// Mitsubishi GX Works2 project: plc   PLC: FX3G

// global labels: Global1
VAR_GLOBAL CONSTANT
  reset_petel_stocks : INT;
END_VAR
VAR_GLOBAL
  petel_stocks AT D2000 : REAL;
  petel_input AT D2500 : REAL;
  lemon_stocks AT D4000 : REAL;
  lemon_input AT D4500 : REAL;
  stabilizer_stocks AT D3000 : REAL;
  stabilizer_input AT D3500 : REAL;
  gummy_stocks AT D5000 : REAL;
  gummy_input AT D5500 : REAL;
  braek_switch AT X005 : BOOL;
  start_switch AT X007 : BOOL;
  valid_input : BOOL;
  start_proces AT X001 : BOOL;
  analog_input AT D8280 : INT;
END_VAR
VAR_GLOBAL CONSTANT
  convert : REAL := 400;
END_VAR
VAR_GLOBAL
  analog_output AT D8282 : INT;
END_VAR
VAR_GLOBAL CONSTANT
  reset_lemonl_stocks : INT;
END_VAR
VAR_GLOBAL
  day_work AT Y007 : BOOL;
  analog_input1_sampled AT M0 : BOOL;
  save_analog_input1 AT D8200 : REAL;
END_VAR
VAR_GLOBAL CONSTANT
  max5 : REAL := 5;
  min6 : REAL := 6;
END_VAR
VAR_GLOBAL
  pinuk_check AT M1 : BOOL;
  regular_check AT M2 : BOOL;
END_VAR
VAR_GLOBAL CONSTANT
  lemon_min_regular : REAL := 455.0;
  petel_min_regular : REAL := 280.0;
  stabilizer_min_regular : REAL := 105.0;
END_VAR
VAR_GLOBAL
  can_make_regular : BOOL;
END_VAR
VAR_GLOBAL CONSTANT
  lemon_min_pinuk : REAL := 655.0;
  petel_min_pinuk : REAL := 385.0;
  stabilizer_min_pinuk : REAL := 210.0;
END_VAR
VAR_GLOBAL
  can_make_pinuk : BOOL;
  make_pinuk AT M4 : BOOL;
  make_regular AT M3 : BOOL;
END_VAR
VAR_GLOBAL CONSTANT
  lemon_for_regular : REAL := 455;
  petel_for_regular : REAL := 280;
  stabilizer_for_regular : REAL := 105;
END_VAR
VAR_GLOBAL
  ready_regular AT M5 : BOOL;
END_VAR
VAR_GLOBAL CONSTANT
  lemon_for_pinuck : REAL := 665;
END_VAR
VAR_GLOBAL
  ready_pinuk AT M6 : BOOL;
END_VAR
VAR_GLOBAL CONSTANT
  petel_for_pinuk : REAL := 385.0;
  stabilizer_for_pinuk : REAL := 210.0;
END_VAR
VAR_GLOBAL
  ice_cream_making AT TC1 : BOOL;
END_VAR
VAR_GLOBAL CONSTANT
  timer_value_5 : INT := 50;
END_VAR
VAR_GLOBAL
  end_making_ice AT TS1 : BOOL;
  making_light AT Y000 : BOOL;
  start_cooling_process AT X002 : BOOL;
  lemon_container AT D6000 : REAL;
  petel_container AT D6300 : REAL;
  petel_cooling_container AT D6800 : REAL;
  lemon_cooling_container AT D7200 : REAL;
  flavors_in_cooling_container AT M7 : BOOL;
  cooling_process_on AT Y002 : BOOL;
END_VAR
VAR_GLOBAL CONSTANT
  timer_value_8 : INT := 80;
END_VAR
VAR_GLOBAL
  temperature_sensor AT X003 : BOOL;
  end_cooling_timer AT TS2 : BOOL;
  cooling_light AT Y002 : BOOL;
  finish_cooling AT M8 : BOOL;
  end_cooling AT Y002 : BOOL;
  mixing_container AT D7400 : REAL;
END_VAR
VAR_GLOBAL CONSTANT
  gummy_for_regular : REAL := 28;
  gummy_for_pinuk : REAL := 70;
END_VAR
VAR_GLOBAL
  pinuk_mixing_starts AT M10 : BOOL;
  regular_mixing_starts AT M9 : BOOL;
  mixing_time_regular AT TC3 : BOOL;
END_VAR
VAR_GLOBAL CONSTANT
  timer_3_sec : INT := 30;
END_VAR
VAR_GLOBAL
  end_mix_regular AT TS3 : BOOL;
  mixing_time_pinuk AT TC4 : BOOL;
END_VAR
VAR_GLOBAL CONSTANT
  timer_5_sec : INT := 50;
END_VAR
VAR_GLOBAL
  end_mix_pinuk AT TS4 : BOOL;
  mixing_process AT M11 : BOOL;
  flicker_y5 AT TC5 : BOOL;
  end_one_flicker_Y5 AT TS5 : BOOL;
END_VAR
VAR_GLOBAL CONSTANT
  timer_flicks : INT := 5;
END_VAR
VAR_GLOBAL
  light_y5 AT Y005 : BOOL;
  flicker_y6 AT TC6 : BOOL;
  end_flicker_y6 AT TS6 : BOOL;
  light_y6 AT Y006 : BOOL;
END_VAR
VAR_GLOBAL CONSTANT
  reset_constant_word : INT := K0;
  reset_constant_float : REAL;
END_VAR
VAR_GLOBAL
  end_mixing_all AT M12 : BOOL;
  start_packing AT X004 : BOOL;
  cup_packaging AT X000 : BOOL;
  cups_counter_7 AT CC1 : BOOL;
END_VAR
VAR_GLOBAL CONSTANT
  gummygam_box : REAL := 1.0;
  converting_to_analong_output : REAL := 40;
END_VAR
VAR_GLOBAL
  packing_light AT Y004 : BOOL;
  cooling_timer AT TC2 : BOOL;
  storage AT D7000 : REAL;
  ice_cream_making_pinuk AT TC7 : BOOL;
  end_making_ice_pinuk AT TS7 : BOOL;
END_VAR
VAR_GLOBAL CONSTANT
  val_6 : INT := 6;
END_VAR
VAR_GLOBAL
  cups_counter AT CS1 : BOOL;
  m_25 AT M25 : BOOL;
  m_26 AT M26 : BOOL;
  m_27 AT M27 : BOOL;
  m_28 AT M28 : BOOL;
  m_29 AT M29 : BOOL;
  m_30 AT M30 : BOOL;
  m_31 AT M31 : BOOL;
  m_32 AT M32 : BOOL;
END_VAR
VAR_GLOBAL CONSTANT
  gummy_min_regular : REAL := 28;
  product_lemon_for_regular : REAL := 525;
  product_petel_for_regular : REAL := 350;
  product_lemon_for_pinuck : REAL := 805;
  product_petel_for_pinuk : REAL := 560;
END_VAR

// task Task_01 (event TRUE, interval 0, priority 31): POU_01

PROGRAM POU_01
(* structured ladder/FBD written out as ST: instructions are called as NAME(EN, inputs, outputs); _pN, _eN, _tN stand for wires *)
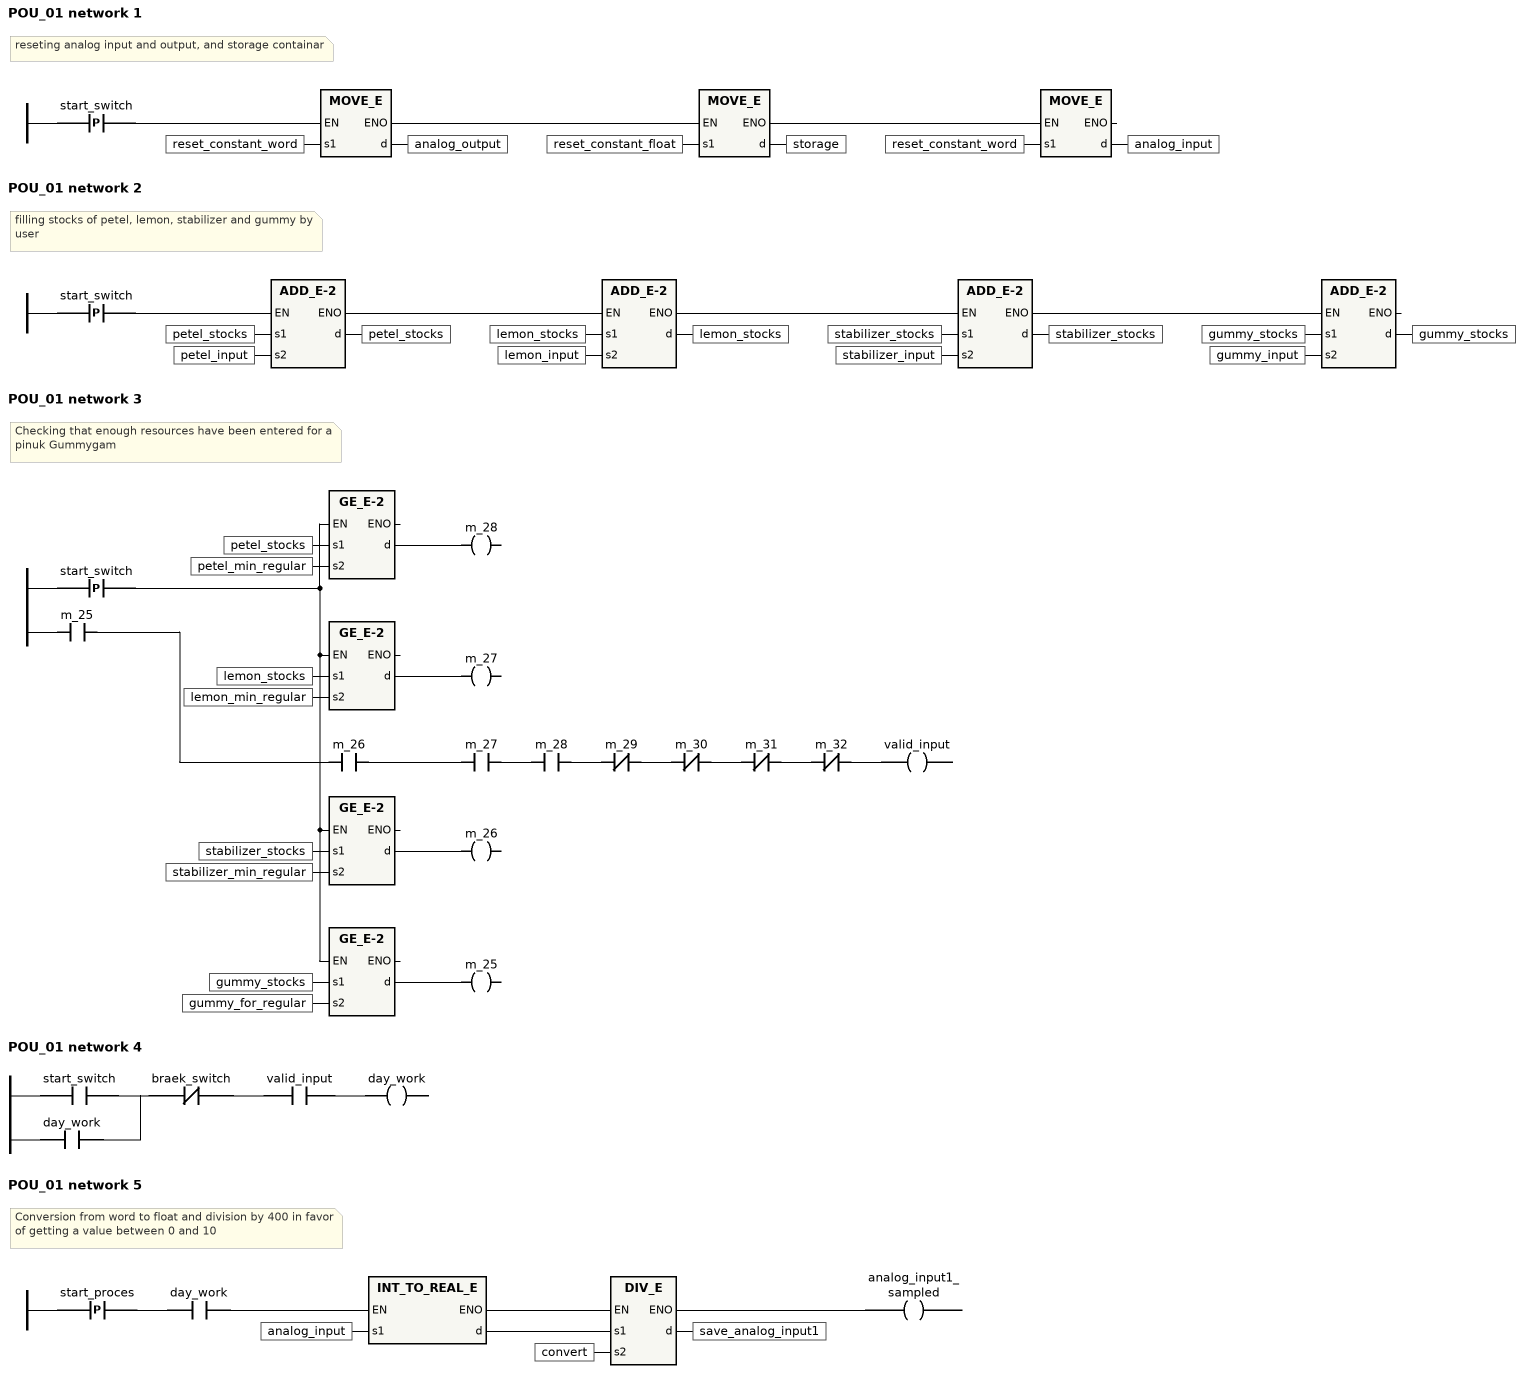
(* network 1 *)
(* reseting analog input and output, and storage containar *)
_e1 := MOVE_E(LDP(TRUE, start_switch), reset_constant_word, analog_output);
_e2 := MOVE_E(_e1, reset_constant_float, storage);
MOVE_E(_e2, reset_constant_word, analog_input);
(* network 2 *)
(* filling stocks of petel, lemon, stabilizer and gummy by user *)
_e1 := ADD_E(LDP(TRUE, start_switch), petel_stocks, petel_input, petel_stocks);
_e2 := ADD_E(_e1, lemon_stocks, lemon_input, lemon_stocks);
_e3 := ADD_E(_e2, stabilizer_stocks, stabilizer_input, stabilizer_stocks);
ADD_E(_e3, gummy_stocks, gummy_input, gummy_stocks);
(* network 3 *)
(* Checking that enough resources have been entered for a pinuk Gummygam *)
_p1 := LDP(TRUE, start_switch);
GE_E(_p1, petel_stocks, petel_min_regular, _t2);
m_28 := _t2;
GE_E(_p1, lemon_stocks, lemon_min_regular, _t3);
m_27 := _t3;
GE_E(_p1, stabilizer_stocks, stabilizer_min_regular, _t4);
m_26 := _t4;
GE_E(_p1, gummy_stocks, gummy_for_regular, _t5);
m_25 := _t5;
valid_input := m_25 AND m_26 AND m_27 AND m_28 AND NOT m_29 AND NOT m_30 AND NOT m_31 AND NOT m_32;
(* network 4 *)
day_work := ((start_switch OR day_work) AND NOT braek_switch) AND valid_input;
(* network 5 *)
(* Conversion from word to float and division by 400 in favor of getting a value between 0 and 10 *)
_e2 := INT_TO_REAL_E(LDP(TRUE, start_proces) AND day_work, analog_input, _t1);
_e3 := DIV_E(_e2, _t1, convert, save_analog_input1);
analog_input1_sampled := _e3;
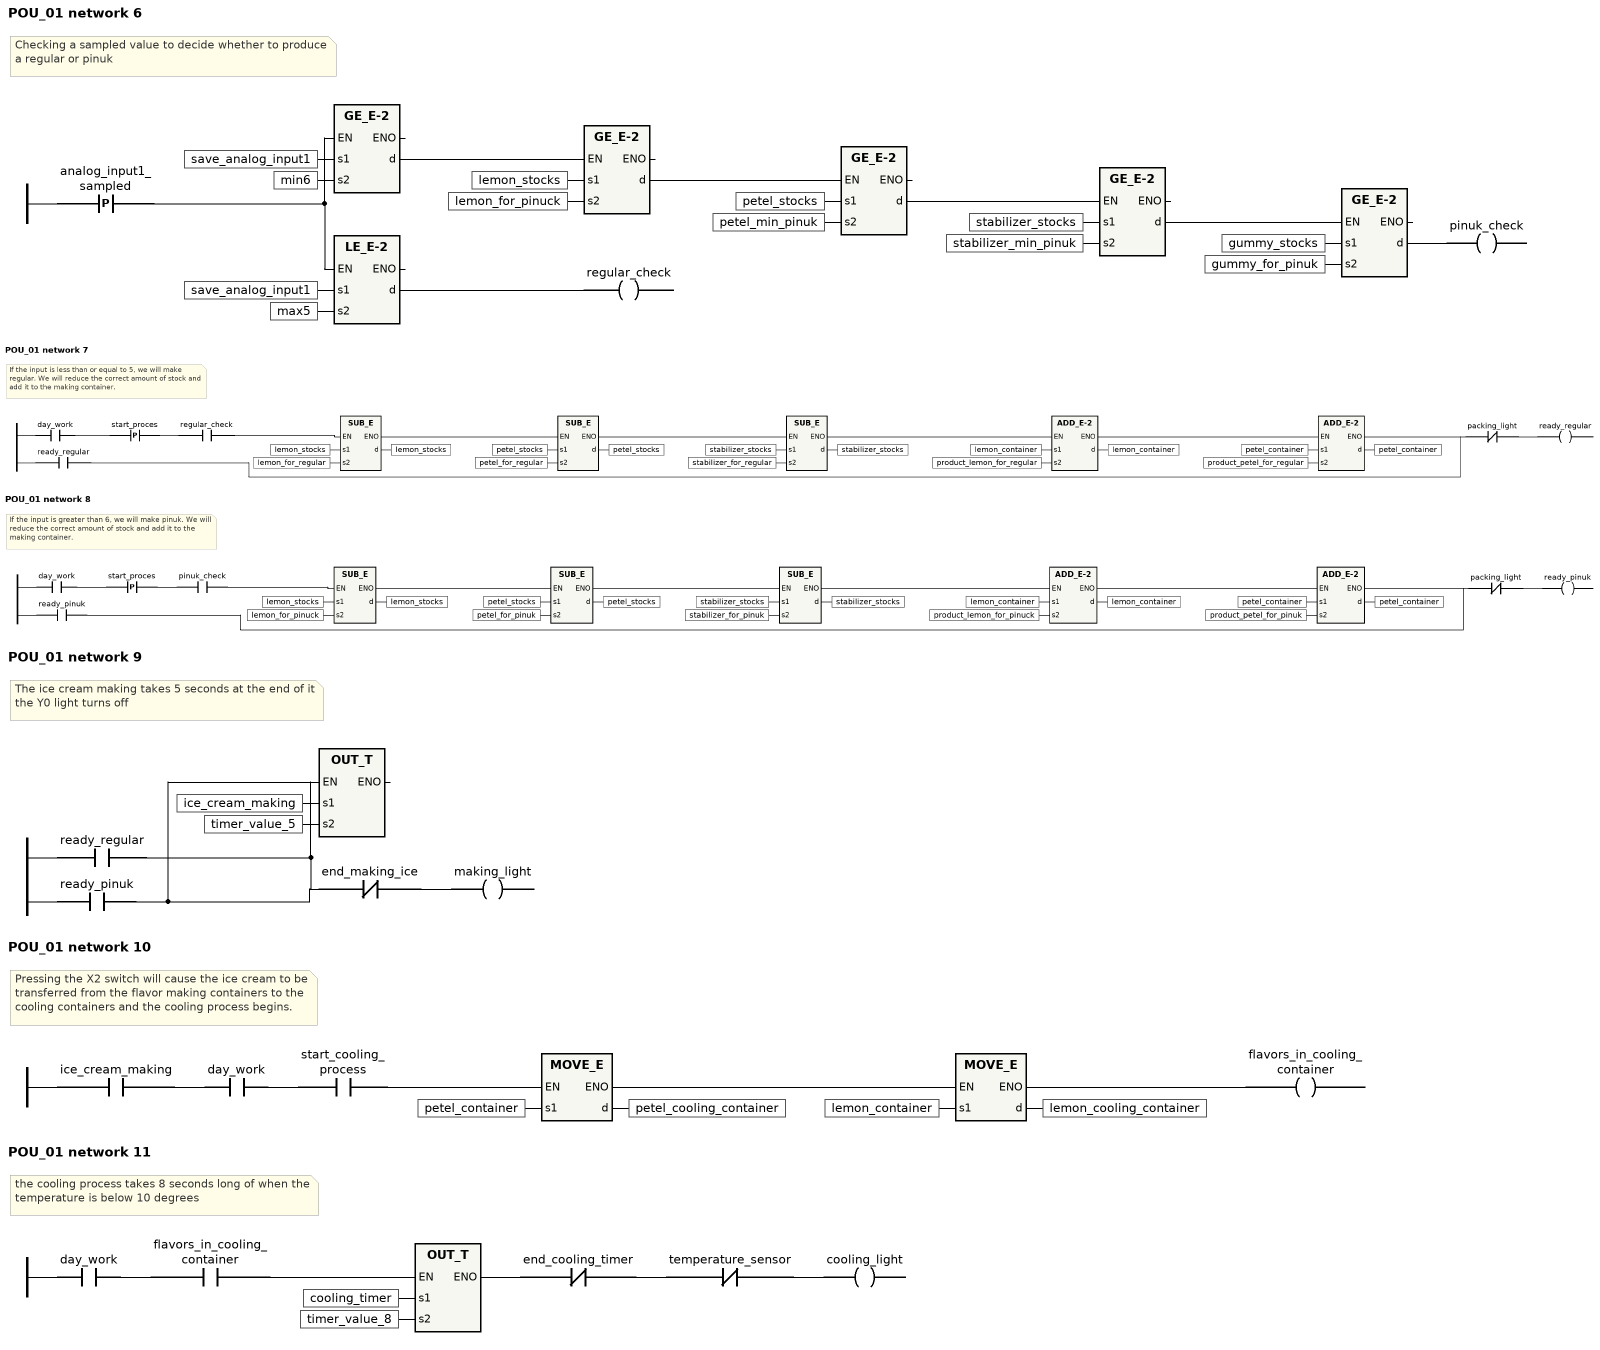
(* network 6 *)
(* Checking a sampled value to decide whether to produce a regular or pinuk *)
_p1 := LDP(TRUE, analog_input1_sampled);
LE_E(_p1, save_analog_input1, max5, _t2);
regular_check := _t2;
GE_E(_p1, save_analog_input1, min6, _t3);
GE_E(_t3, lemon_stocks, lemon_for_pinuck, _t4);
GE_E(_t4, petel_stocks, petel_min_pinuk, _t5);
GE_E(_t5, stabilizer_stocks, stabilizer_min_pinuk, _t6);
GE_E(_t6, gummy_stocks, gummy_for_pinuk, _t7);
pinuk_check := _t7;
(* network 7 *)
(* If the input is less than or equal to 5, we will make regular. We will reduce the correct amount of stock and add it to the making container. *)
_e1 := SUB_E(day_work AND LDP(TRUE, start_proces) AND regular_check, lemon_stocks, lemon_for_regular, lemon_stocks);
_e2 := SUB_E(_e1, petel_stocks, petel_for_regular, petel_stocks);
_e3 := SUB_E(_e2, stabilizer_stocks, stabilizer_for_regular, stabilizer_stocks);
_e4 := ADD_E(_e3, lemon_container, product_lemon_for_regular, lemon_container);
_e5 := ADD_E(_e4, petel_container, product_petel_for_regular, petel_container);
ready_regular := (_e5 OR ready_regular) AND NOT packing_light;
(* network 8 *)
(* If the input is greater than 6, we will make pinuk. We will reduce the correct amount of stock and add it to the making container. *)
_e1 := SUB_E(day_work AND LDP(TRUE, start_proces) AND pinuk_check, lemon_stocks, lemon_for_pinuck, lemon_stocks);
_e2 := SUB_E(_e1, petel_stocks, petel_for_pinuk, petel_stocks);
_e3 := SUB_E(_e2, stabilizer_stocks, stabilizer_for_pinuk, stabilizer_stocks);
_e4 := ADD_E(_e3, lemon_container, product_lemon_for_pinuck, lemon_container);
_e5 := ADD_E(_e4, petel_container, product_petel_for_pinuk, petel_container);
ready_pinuk := (_e5 OR ready_pinuk) AND NOT packing_light;
(* network 9 *)
(* The ice cream making takes 5 seconds at the end of it the Y0 light turns off *)
_p1 := ready_regular OR ready_pinuk;
OUT_T(_p1, ice_cream_making, timer_value_5);
making_light := _p1 AND NOT end_making_ice;
(* network 10 *)
(* Pressing the X2 switch will cause the ice cream to be transferred from the flavor making containers to the cooling containers and the cooling process begins. *)
_e1 := MOVE_E(ice_cream_making AND day_work AND start_cooling_process, petel_container, petel_cooling_container);
_e2 := MOVE_E(_e1, lemon_container, lemon_cooling_container);
flavors_in_cooling_container := _e2;
(* network 11 *)
(* the cooling process takes 8 seconds long of when the temperature is below 10 degrees *)
_e1 := OUT_T(day_work AND flavors_in_cooling_container, cooling_timer, timer_value_8);
cooling_light := _e1 AND NOT end_cooling_timer AND NOT temperature_sensor;
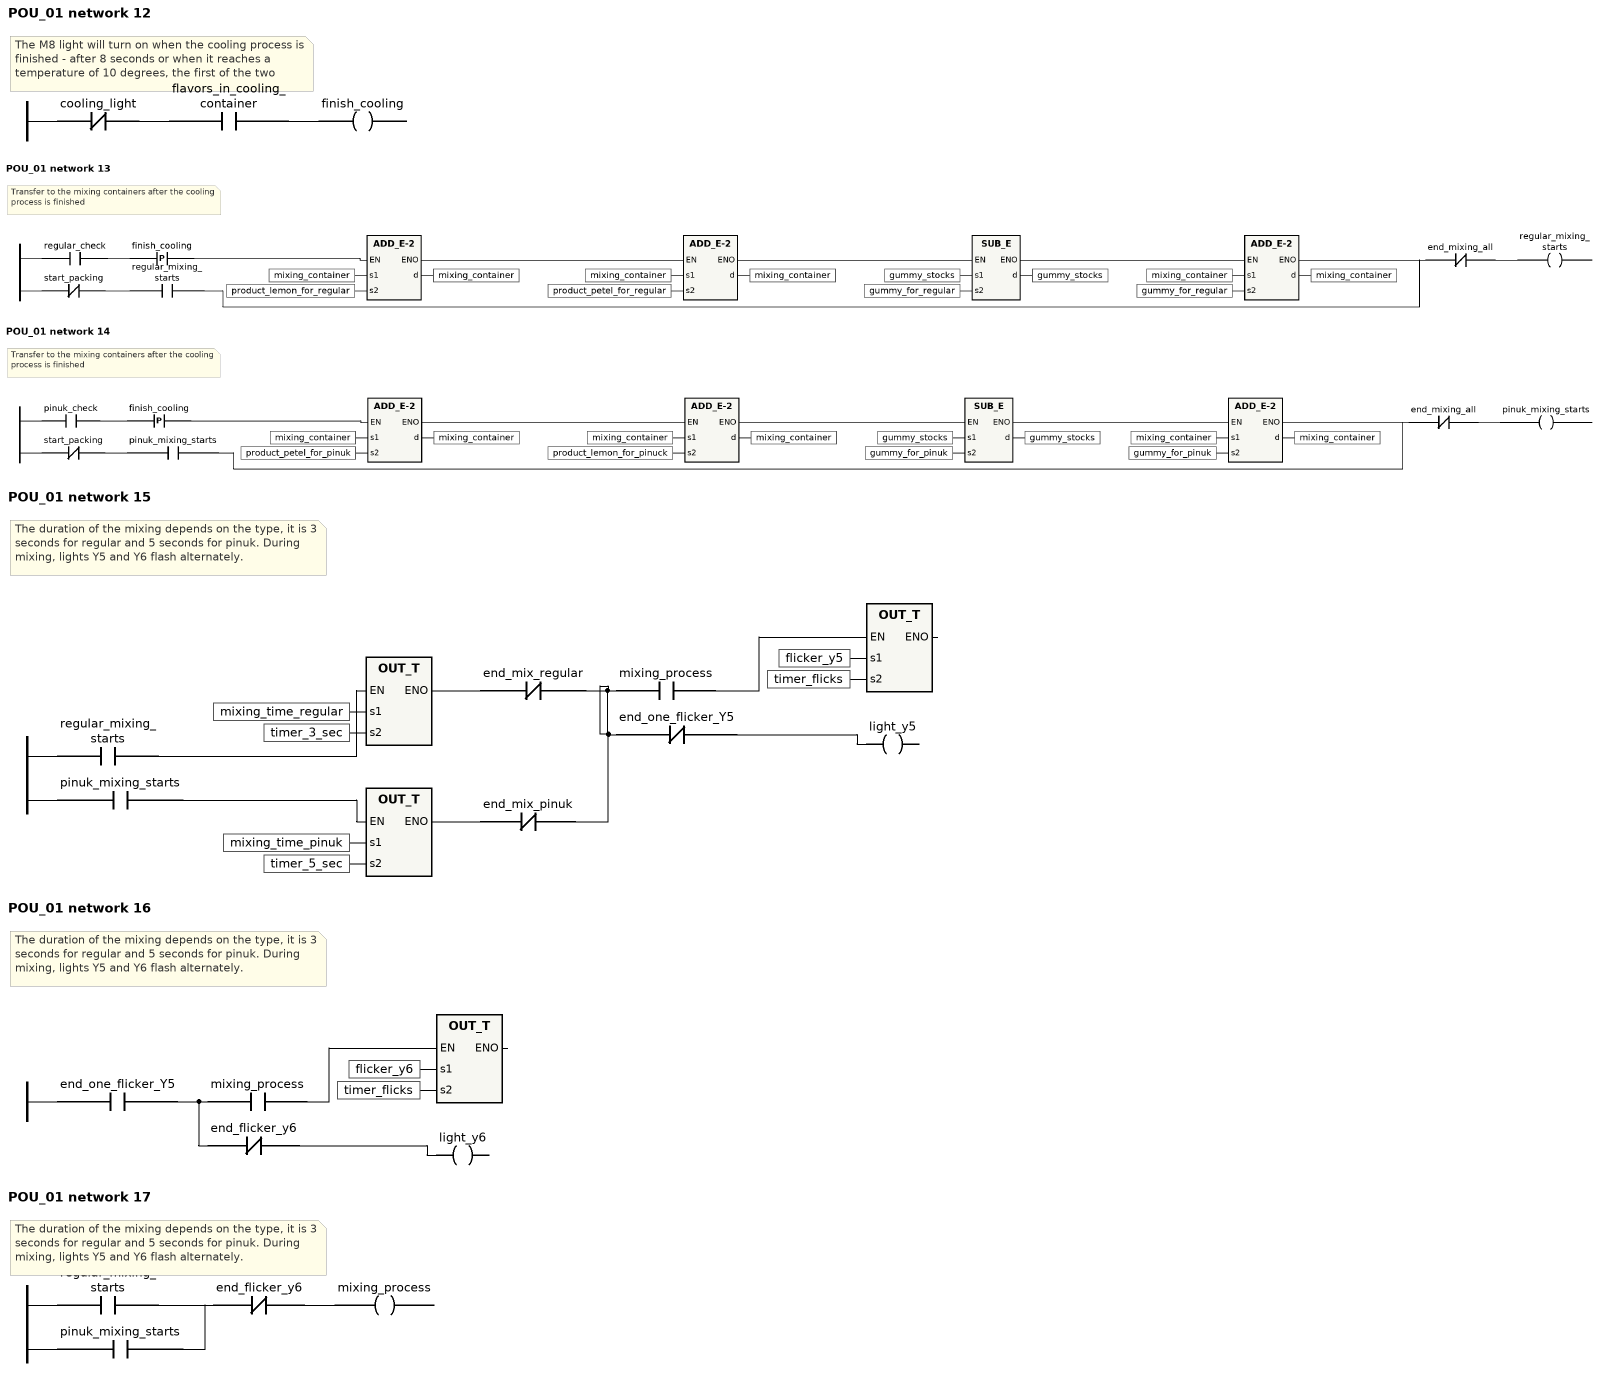
(* network 12 *)
(* The M8 light will turn on when the cooling process is finished - after 8 seconds or when it reaches a temperature of 10 degrees, the first of the two *)
finish_cooling := NOT cooling_light AND flavors_in_cooling_container;
(* network 13 *)
(* Transfer to the mixing containers after the cooling process is finished *)
_e1 := ADD_E(regular_check AND LDP(TRUE, finish_cooling), mixing_container, product_lemon_for_regular, mixing_container);
_e2 := ADD_E(_e1, mixing_container, product_petel_for_regular, mixing_container);
_e3 := SUB_E(_e2, gummy_stocks, gummy_for_regular, gummy_stocks);
_e4 := ADD_E(_e3, mixing_container, gummy_for_regular, mixing_container);
regular_mixing_starts := (_e4 OR (NOT start_packing AND regular_mixing_starts)) AND NOT end_mixing_all;
(* network 14 *)
(* Transfer to the mixing containers after the cooling process is finished *)
_e1 := ADD_E(pinuk_check AND LDP(TRUE, finish_cooling), mixing_container, product_petel_for_pinuk, mixing_container);
_e2 := ADD_E(_e1, mixing_container, product_lemon_for_pinuck, mixing_container);
_e3 := SUB_E(_e2, gummy_stocks, gummy_for_pinuk, gummy_stocks);
_e4 := ADD_E(_e3, mixing_container, gummy_for_pinuk, mixing_container);
pinuk_mixing_starts := (_e4 OR (NOT start_packing AND pinuk_mixing_starts)) AND NOT end_mixing_all;
(* network 15 *)
(* The duration of the mixing depends on the type, it is 3 seconds for regular and 5 seconds for pinuk. During mixing, lights Y5 and Y6 flash alternately. *)
_e1 := OUT_T(regular_mixing_starts, mixing_time_regular, timer_3_sec);
_e2 := OUT_T(pinuk_mixing_starts, mixing_time_pinuk, timer_5_sec);
_p3 := (_e1 AND NOT end_mix_regular) OR (_e2 AND NOT end_mix_pinuk);
OUT_T(_p3 AND mixing_process, flicker_y5, timer_flicks);
light_y5 := _p3 AND NOT end_one_flicker_Y5;
(* network 16 *)
(* The duration of the mixing depends on the type, it is 3 seconds for regular and 5 seconds for pinuk. During mixing, lights Y5 and Y6 flash alternately. *)
OUT_T(end_one_flicker_Y5 AND mixing_process, flicker_y6, timer_flicks);
light_y6 := end_one_flicker_Y5 AND NOT end_flicker_y6;
(* network 17 *)
(* The duration of the mixing depends on the type, it is 3 seconds for regular and 5 seconds for pinuk. During mixing, lights Y5 and Y6 flash alternately. *)
mixing_process := (regular_mixing_starts OR pinuk_mixing_starts) AND NOT end_flicker_y6;
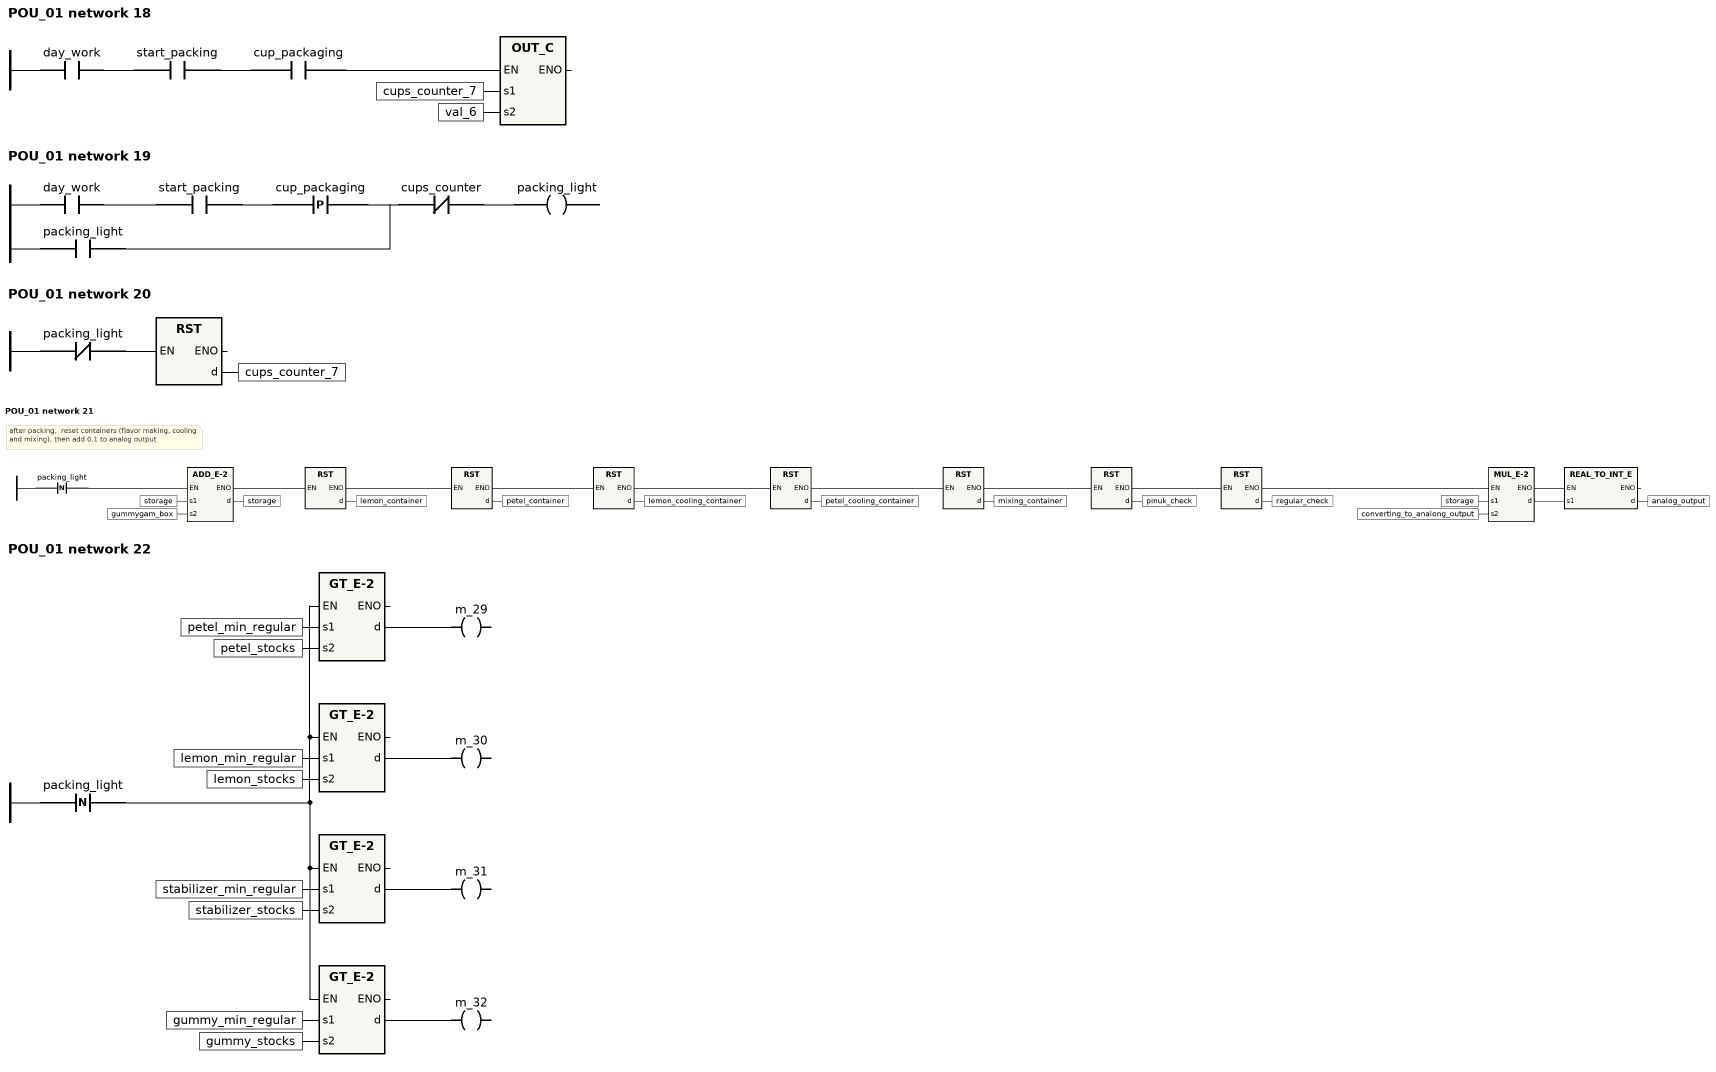
(* network 18 *)
OUT_C(day_work AND start_packing AND cup_packaging, cups_counter_7, val_6);
(* network 19 *)
packing_light := ((day_work AND start_packing AND LDP(TRUE, cup_packaging)) OR packing_light) AND NOT cups_counter;
(* network 20 *)
RST(NOT packing_light, cups_counter_7);
(* network 21 *)
(* after packing,  reset containers (flavor making, cooling and mixing), then add 0.1 to analog output *)
_e1 := ADD_E(LDF(TRUE, packing_light), storage, gummygam_box, storage);
_e2 := RST(_e1, lemon_container);
_e3 := RST(_e2, petel_container);
_e4 := RST(_e3, lemon_cooling_container);
_e5 := RST(_e4, petel_cooling_container);
_e6 := RST(_e5, mixing_container);
_e7 := RST(_e6, pinuk_check);
_e8 := RST(_e7, regular_check);
_e10 := MUL_E(_e8, storage, converting_to_analong_output, _t9);
REAL_TO_INT_E(_e10, _t9, analog_output);
(* network 22 *)
_p1 := LDF(TRUE, packing_light);
GT_E(_p1, petel_min_regular, petel_stocks, _t2);
m_29 := _t2;
GT_E(_p1, lemon_min_regular, lemon_stocks, _t3);
m_30 := _t3;
GT_E(_p1, stabilizer_min_regular, stabilizer_stocks, _t4);
m_31 := _t4;
GT_E(_p1, gummy_min_regular, gummy_stocks, _t5);
m_32 := _t5;
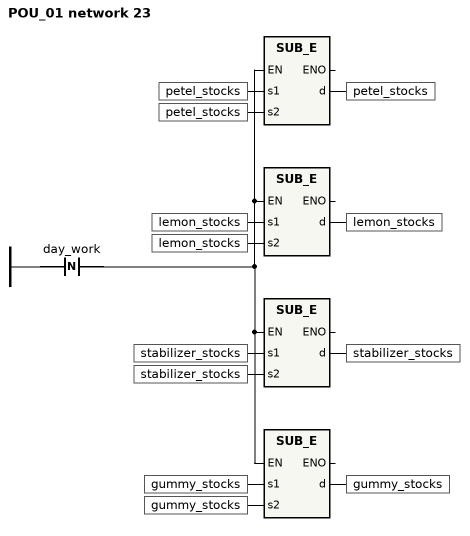
(* network 23 *)
_p1 := LDF(TRUE, day_work);
SUB_E(_p1, petel_stocks, petel_stocks, petel_stocks);
SUB_E(_p1, lemon_stocks, lemon_stocks, lemon_stocks);
SUB_E(_p1, stabilizer_stocks, stabilizer_stocks, stabilizer_stocks);
SUB_E(_p1, gummy_stocks, gummy_stocks, gummy_stocks);
END_PROGRAM
